{attribute addProperty BoxType "EJ9576-0000-0020"}
{attribute addProperty Id "BCT_InputsAT %I*BCT_Inputs_047F8208128160WcStateAT %I*WcState_F855686C1620InfoDataAT %I*InfoData_BC63D37F80100"}
{attribute addProperty CRC "2602112332"}
{attribute addProperty SizeInBites "224"}
{attribute addProperty SizeInBytes "28"}
TYPE EJ9576_57CA9E36 :
STRUCT
	{attribute addProperty Name "BCT_Inputs"}
	BCT_Inputs : BCT_Inputs_047F8208;
	{attribute addProperty Name "WcState"}
	WcState : WcState_F855686C;
	{attribute addProperty Name "InfoData"}
	InfoData : InfoData_BC63D37F;
END_STRUCT
END_TYPE

(* stored: Version 1.2.0.0, ProductVersion 3.1.4024.9
   DUT EJ9576_57CA9E36: Id {8ef56fd7-3d5a-4c4a-b905-50902a32ba4a} *)
